{attribute 'qualified_only'}
VAR_GLOBAL	
	{attribute 'OPC.UA.DA.StructuredType' := '1'}
	sTurnTable: Turntable;
	sRollerConveyor: RollerConveyor;
	
	{attribute 'OPC.UA.DA' := '1'}
	bDiffuseSensorPaletA	:BOOL;
	{attribute 'OPC.UA.DA' := '1'}
	bDiffuseSensorPaletV	:BOOL;
	{attribute 'OPC.UA.DA' := '1'}
	bDiffuseSensorPaletM	:BOOL;
	{attribute 'OPC.UA.DA' := '1'}	
	bVisionSensorSalida		:DINT;
	
	{attribute 'OPC.UA.DA' := '1'}
	iLightArrayEmitterA		:BOOL;
	{attribute 'OPC.UA.DA' := '1'}
	iLightArrayEmitterV		:BOOL;
	{attribute 'OPC.UA.DA' := '1'}
	iLightArrayEmitterM		:BOOL; 
END_VAR

(* stored: Version 1.1.0.1, ProductVersion 3.1.4024.12
   GVL GVL_ProcesoPalet: Id {ed6e88b2-2b23-44c0-8618-d50017000d77} *)
